PROGRAM AxisAbs
VAR
	nSpeed_MoveAbs						:LREAL:=5;
	
	nTargetPos_MoveAbs								:LREAL;

END_VAR


// LeftArm_Left_MoveAbs
IF bManualCtrl_Part_LeftArm_Left THEN					
	axis_LeftArm_Left_MoveAbs(
		Axis:= axis_LeftArm_Left, 
		Execute:= bAxis_LeftArm_Left_MoveAbs, 
		Position:= nTargetPos_MoveAbs, 
		Velocity:= nSpeed_MoveAbs, 
		Acceleration:= , 
		Deceleration:= , 
		Jerk:= , 
		BufferMode:= , 
		Options:= , 
		Done=> , 
		Busy=> , 
		Active=> , 
		CommandAborted=> , 
		Error=> , 
		ErrorID=> );	
END_IF

// LeftArm_Right_MoveAbs
IF bManualCtrl_Part_LeftArm_Right THEN					
	axis_LeftArm_Right_MoveAbs(
		Axis:= axis_LeftArm_Right, 
		Execute:= bAxis_LeftArm_Right_MoveAbs, 
		Position:= nTargetPos_MoveAbs, 
		Velocity:= nSpeed_MoveAbs, 
		Acceleration:= , 
		Deceleration:= , 
		Jerk:= , 
		BufferMode:= , 
		Options:= , 
		Done=> , 
		Busy=> , 
		Active=> , 
		CommandAborted=> , 
		Error=> , 
		ErrorID=> );	
END_IF


// LeftArm_Wrist_MoveAbs
IF bManualCtrl_Part_LeftArm_Wrist THEN					
	axis_LeftArm_Wrist_MoveAbs(
		Axis:= axis_LeftArm_Wrist, 
		Execute:= bAxis_LeftArm_Wrist_MoveAbs, 
		Position:= nTargetPos_MoveAbs, 
		Velocity:= nSpeed_MoveAbs, 
		Acceleration:= , 
		Deceleration:= , 
		Jerk:= , 
		BufferMode:= , 
		Options:= , 
		Done=> , 
		Busy=> , 
		Active=> , 
		CommandAborted=> , 
		Error=> , 
		ErrorID=> );	
END_IF


// LeftArm_Lift_MoveAbs
IF bManualCtrl_Part_LeftArm_Lift THEN					
	axis_LeftArm_Lift_MoveAbs(
		Axis:= axis_LeftArm_Lift, 
		Execute:= bAxis_LeftArm_Lift_MoveAbs, 
		Position:= nTargetPos_MoveAbs, 
		Velocity:= nSpeed_MoveAbs, 
		Acceleration:= , 
		Deceleration:= , 
		Jerk:= , 
		BufferMode:= , 
		Options:= , 
		Done=> , 
		Busy=> , 
		Active=> , 
		CommandAborted=> , 
		Error=> , 
		ErrorID=> );	
END_IF



// RightArm_Left_MoveAbs
IF bManualCtrl_Part_RightArm_Left THEN					
	axis_RightArm_Left_MoveAbs(
		Axis:= axis_RightArm_Left, 
		Execute:= bAxis_RightArm_Left_MoveAbs, 
		Position:= nTargetPos_MoveAbs, 
		Velocity:= nSpeed_MoveAbs, 
		Acceleration:= , 
		Deceleration:= , 
		Jerk:= , 
		BufferMode:= , 
		Options:= , 
		Done=> , 
		Busy=> , 
		Active=> , 
		CommandAborted=> , 
		Error=> , 
		ErrorID=> );	
END_IF

// RightArm_Right_MoveAbs
IF bManualCtrl_Part_RightArm_Right THEN					
	axis_RightArm_Right_MoveAbs(
		Axis:= axis_RightArm_Right, 
		Execute:= bAxis_RightArm_Right_MoveAbs, 
		Position:= nTargetPos_MoveAbs, 
		Velocity:= nSpeed_MoveAbs, 
		Acceleration:= , 
		Deceleration:= , 
		Jerk:= , 
		BufferMode:= , 
		Options:= , 
		Done=> , 
		Busy=> , 
		Active=> , 
		CommandAborted=> , 
		Error=> , 
		ErrorID=> );	
END_IF


// RightArm_Wrist_MoveAbs
IF bManualCtrl_Part_RightArm_Wrist THEN					
	axis_RightArm_Wrist_MoveAbs(
		Axis:= axis_RightArm_Wrist, 
		Execute:= bAxis_RightArm_Wrist_MoveAbs, 
		Position:= nTargetPos_MoveAbs, 
		Velocity:= nSpeed_MoveAbs, 
		Acceleration:= , 
		Deceleration:= , 
		Jerk:= , 
		BufferMode:= , 
		Options:= , 
		Done=> , 
		Busy=> , 
		Active=> , 
		CommandAborted=> , 
		Error=> , 
		ErrorID=> );	
END_IF


// RightArm_Lift_MoveAbs
IF bManualCtrl_Part_RightArm_Lift THEN					
	axis_RightArm_Lift_MoveAbs(
		Axis:= axis_RightArm_Lift, 
		Execute:= bAxis_RightArm_Lift_MoveAbs, 
		Position:= nTargetPos_MoveAbs, 
		Velocity:= nSpeed_MoveAbs, 
		Acceleration:= , 
		Deceleration:= , 
		Jerk:= , 
		BufferMode:= , 
		Options:= , 
		Done=> , 
		Busy=> , 
		Active=> , 
		CommandAborted=> , 
		Error=> , 
		ErrorID=> );	
END_IF


// BigGate_Left_MoveAbs
IF bManualCtrl_Part_BigGate_Left THEN					
	axis_BigGate_Left_MoveAbs(
		Axis:= axis_BigGate_Left, 
		Execute:= bAxis_BigGate_Left_MoveAbs, 
		Position:= nTargetPos_MoveAbs, 
		Velocity:= nSpeed_MoveAbs, 
		Acceleration:= , 
		Deceleration:= , 
		Jerk:= , 
		BufferMode:= , 
		Options:= , 
		Done=> , 
		Busy=> , 
		Active=> , 
		CommandAborted=> , 
		Error=> , 
		ErrorID=> );	
END_IF

// BigGate_Right_MoveAbs
IF bManualCtrl_Part_BigGate_Right THEN					
	axis_BigGate_Right_MoveAbs(
		Axis:= axis_BigGate_Right, 
		Execute:= bAxis_BigGate_Right_MoveAbs, 
		Position:= nTargetPos_MoveAbs, 
		Velocity:= nSpeed_MoveAbs, 
		Acceleration:= , 
		Deceleration:= , 
		Jerk:= , 
		BufferMode:= , 
		Options:= , 
		Done=> , 
		Busy=> , 
		Active=> , 
		CommandAborted=> , 
		Error=> , 
		ErrorID=> );	
END_IF

// SmallGate_Left_MoveAbs
IF bManualCtrl_Part_SmallGate_Left THEN					
	axis_SmallGate_Left_MoveAbs(
		Axis:= axis_SmallGate_Left, 
		Execute:= bAxis_SmallGate_Left_MoveAbs, 
		Position:= nTargetPos_MoveAbs, 
		Velocity:= nSpeed_MoveAbs, 
		Acceleration:= , 
		Deceleration:= , 
		Jerk:= , 
		BufferMode:= , 
		Options:= , 
		Done=> , 
		Busy=> , 
		Active=> , 
		CommandAborted=> , 
		Error=> , 
		ErrorID=> );	
END_IF

// SmallGate_Right_MoveAbs
IF bManualCtrl_Part_SmallGate_Right THEN					
	axis_SmallGate_Right_MoveAbs(
		Axis:= axis_SmallGate_Right, 
		Execute:= bAxis_SmallGate_Right_MoveAbs, 
		Position:= nTargetPos_MoveAbs, 
		Velocity:= nSpeed_MoveAbs, 
		Acceleration:= , 
		Deceleration:= , 
		Jerk:= , 
		BufferMode:= , 
		Options:= , 
		Done=> , 
		Busy=> , 
		Active=> , 
		CommandAborted=> , 
		Error=> , 
		ErrorID=> );	
END_IF


// BackGate_Left_MoveAbs
IF bManualCtrl_Part_BackGate_Left THEN					
	axis_BackGate_Left_MoveAbs(
		Axis:= axis_BackGate_Left, 
		Execute:= bAxis_BackGate_Left_MoveAbs, 
		Position:= nTargetPos_MoveAbs, 
		Velocity:= nSpeed_MoveAbs, 
		Acceleration:= , 
		Deceleration:= , 
		Jerk:= , 
		BufferMode:= , 
		Options:= , 
		Done=> , 
		Busy=> , 
		Active=> , 
		CommandAborted=> , 
		Error=> , 
		ErrorID=> );	
END_IF

// BackGate_Right_MoveAbs
IF bManualCtrl_Part_BackGate_Right THEN					
	axis_BackGate_Right_MoveAbs(
		Axis:= axis_BackGate_Right, 
		Execute:= bAxis_BackGate_Right_MoveAbs, 
		Position:= nTargetPos_MoveAbs, 
		Velocity:= nSpeed_MoveAbs, 
		Acceleration:= , 
		Deceleration:= , 
		Jerk:= , 
		BufferMode:= , 
		Options:= , 
		Done=> , 
		Busy=> , 
		Active=> , 
		CommandAborted=> , 
		Error=> , 
		ErrorID=> );	
END_IF

END_PROGRAM

(* stored: Version 1.1.0.1, ProductVersion 3.1.4024.14
   POU AxisAbs: Id {e09c7cd3-7a67-4bf0-8215-dcda5e249eef}, SpecialFunc None *)
